   cmMendrelCathodeFrontAxisY.commandConfiguration.offset.offset := 0.0;
   cmMendrelCathodeFrontAxisY.commandConfiguration.offset.profileReference := 1;
   cmMendrelCathodeFrontAxisY.commandConfiguration.offset.offsetDistance := 0.0;
   cmMendrelCathodeFrontAxisY.commandConfiguration.offset.startPosition := 0.0;
   cmMendrelCathodeFrontAxisY.commandConfiguration.offset.direction := 3;
   cmMendrelCathodeFrontAxisY.commandConfiguration.offset.offsetAbsolute := TRUE;
   cmMendrelCathodeFrontAxisY.commandConfiguration.offset.offsetChangeOnTheFly := FALSE;
   cmMendrelCathodeFrontAxisY.commands.enableAxis := FALSE;
   cmMendrelCathodeFrontAxisY.commands.resetAxis := FALSE;
   cmMendrelCathodeFrontAxisY.commands.openBrake := FALSE;
   cmMendrelCathodeFrontAxisY.commands.jogForward := FALSE;
   cmMendrelCathodeFrontAxisY.commands.jogBackward := FALSE;
   cmMendrelCathodeFrontAxisY.commands.moveVelocity := FALSE;
   cmMendrelCathodeFrontAxisY.commands.stop := FALSE;
   cmMendrelCathodeFrontAxisY.commands.fastStop := FALSE;
   cmMendrelCathodeFrontAxisY.commands.torqueLimiting := FALSE;
   cmMendrelCathodeFrontAxisY.commands.homing := FALSE;
   cmMendrelCathodeFrontAxisY.commands.posRelative := FALSE;
   cmMendrelCathodeFrontAxisY.commands.posAbsolute := FALSE;
   cmMendrelCathodeFrontAxisY.commands.posSuperimposed := FALSE;
   cmMendrelCathodeFrontAxisY.commands.haltSuperimposed := FALSE;
   cmMendrelCathodeFrontAxisY.commands.selectSetPosition := -1;
   cmMendrelCathodeFrontAxisY.commands.reset := FALSE;
   cmMendrelCathodeFrontAxisY.monitoring.valid := FALSE;
   cmMendrelCathodeFrontAxisY.monitoring.busy := TRUE;
   cmMendrelCathodeFrontAxisY.monitoring.error := TRUE;
   cmMendrelCathodeFrontAxisY.monitoring.status := 16#8600;
   cmMendrelCathodeFrontAxisY.monitoring.subfunctionStatus := 16#8001;
   cmMendrelCathodeFrontAxisY.monitoring.axisEnabled := FALSE;
   cmMendrelCathodeFrontAxisY.monitoring.resetActive := FALSE;
   cmMendrelCathodeFrontAxisY.monitoring.inVelocity := FALSE;
   cmMendrelCathodeFrontAxisY.monitoring.inLimitation := FALSE;
   cmMendrelCathodeFrontAxisY.monitoring.inClamping := FALSE;
   cmMendrelCathodeFrontAxisY.monitoring.startSync := FALSE;
   cmMendrelCathodeFrontAxisY.monitoring.inSync := FALSE;
   cmMendrelCathodeFrontAxisY.monitoring.inSimulation := FALSE;
   cmMendrelCathodeFrontAxisY.monitoring.jogSelected := FALSE;
   cmMendrelCathodeFrontAxisY.monitoring.moveVelocitySelected := FALSE;
   cmMendrelCathodeFrontAxisY.monitoring.stopSelected := FALSE;
   cmMendrelCathodeFrontAxisY.monitoring.fastStopSelected := FALSE;
   cmMendrelCathodeFrontAxisY.monitoring.torqueLimitingSelected := FALSE;
   cmMendrelCathodeFrontAxisY.monitoring.homingSelected := FALSE;
   cmMendrelCathodeFrontAxisY.monitoring.posRelativeSelected := FALSE;
   cmMendrelCathodeFrontAxisY.monitoring.posAbsoluteSelected := FALSE;
   cmMendrelCathodeFrontAxisY.monitoring.posSuperimposedSelected := FALSE;
   cmMendrelCathodeFrontAxisY.monitoring.haltSuperimposedSelected := FALSE;
   cmMendrelCathodeFrontAxisY.monitoring.commandBusy := FALSE;
   cmMendrelCathodeFrontAxisY.monitoring.commandDone := FALSE;
   cmMendrelCathodeFrontAxisY.monitoring.commandAborted := FALSE;
   cmMendrelCathodeFrontAxisY.monitoring.homingCommandBusy := FALSE;
   cmMendrelCathodeFrontAxisY.monitoring.homingCommandDone := FALSE;
   cmMendrelCathodeFrontAxisY.monitoring.homingCommandAborted := FALSE;
   cmMendrelCathodeFrontAxisY.monitoring.superimposedBusy := FALSE;
   cmMendrelCathodeFrontAxisY.monitoring.superimposedDone := FALSE;
   cmMendrelCathodeFrontAxisY.monitoring.superimposedAborted := FALSE;
   cmMendrelCathodeFrontAxisY.monitoring.actualPosition := 10.963;
   cmMendrelCathodeFrontAxisY.monitoring.actualSpeed := 0.0;
   cmMendrelCathodeFrontAxisY.monitoring.speedUnit := 1062;
   cmMendrelCathodeFrontAxisY.monitoring.positionUnit := 1013;
   cmMendrelCathodeFrontAxisY.monitoring.axisType := 1;
   cmMendrelCathodeFrontAxisY.monitoring.interlockGeneralOut := TRUE;
   cmMendrelCathodeFrontAxisY.monitoring.interlockJogForwardOut := TRUE;
   cmMendrelCathodeFrontAxisY.monitoring.interlockJogBackwardOut := TRUE;
   cmMendrelCathodeFrontAxisZ.commandConfiguration.generalSettings.stopOnError := TRUE;
   cmMendrelCathodeFrontAxisZ.commandConfiguration.generalSettings.resetWithRestart := FALSE;
   cmMendrelCathodeFrontAxisZ.commandConfiguration.generalSettings.abortWaitingSyncCmd := TRUE;
   cmMendrelCathodeFrontAxisZ.commandConfiguration.power.startMode := 1;
   cmMendrelCathodeFrontAxisZ.commandConfiguration.power.stopMode := 0;
   cmMendrelCathodeFrontAxisZ.commandConfiguration.power.syncMotionSimulation := FALSE;
   cmMendrelCathodeFrontAxisZ.commandConfiguration.power.syncMotionSimulationExtendedMode := -1;
   cmMendrelCathodeFrontAxisZ.commandConfiguration.jog.velocity := 5.0;
   cmMendrelCathodeFrontAxisZ.commandConfiguration.jog.acceleration := 50.0;
   cmMendrelCathodeFrontAxisZ.commandConfiguration.jog.deceleration := 50.0;
   cmMendrelCathodeFrontAxisZ.commandConfiguration.jog.jerk := -1.0;
   cmMendrelCathodeFrontAxisZ.commandConfiguration.jog.positionControlled := TRUE;
   cmMendrelCathodeFrontAxisZ.commandConfiguration.jog.increment := 0.0;
   cmMendrelCathodeFrontAxisZ.commandConfiguration.jog.mode := 0;
   cmMendrelCathodeFrontAxisZ.commandConfiguration.moveVelocity.velocity := 0.0;
   cmMendrelCathodeFrontAxisZ.commandConfiguration.moveVelocity.acceleration := -1.0;
   cmMendrelCathodeFrontAxisZ.commandConfiguration.moveVelocity.deceleration := -1.0;
   cmMendrelCathodeFrontAxisZ.commandConfiguration.moveVelocity.jerk := -1.0;
   cmMendrelCathodeFrontAxisZ.commandConfiguration.moveVelocity.direction := 0;
   cmMendrelCathodeFrontAxisZ.commandConfiguration.moveVelocity.positionControlled := TRUE;
   cmMendrelCathodeFrontAxisZ.commandConfiguration.moveVelocity.velocityChangeOnTheFly := FALSE;
   cmMendrelCathodeFrontAxisZ.commandConfiguration.stop.deceleration := -1.0;
   cmMendrelCathodeFrontAxisZ.commandConfiguration.stop.jerk := -1.0;
   cmMendrelCathodeFrontAxisZ.commandConfiguration.stop.abortAcceleration := FALSE;
   cmMendrelCathodeFrontAxisZ.commandConfiguration.fastStop.deceleration := -1.0;
   cmMendrelCathodeFrontAxisZ.commandConfiguration.fastStop.jerk := -1.0;
   cmMendrelCathodeFrontAxisZ.commandConfiguration.fastStop.abortAcceleration := FALSE;
   cmMendrelCathodeFrontAxisZ.commandConfiguration.fastStop.replaceStopPossible := FALSE;
   cmMendrelCathodeFrontAxisZ.commandConfiguration.torqueLimiting.limit := -1.0;
   cmMendrelCathodeFrontAxisZ.commandConfiguration.torqueLimiting.mode := 0;
   cmMendrelCathodeFrontAxisZ.commandConfiguration.homing.position := 0.0;
   cmMendrelCathodeFrontAxisZ.commandConfiguration.homing.mode := 0;
   cmMendrelCathodeFrontAxisZ.commandConfiguration.homing.sensor := 0;
   cmMendrelCathodeFrontAxisZ.commandConfiguration.homing.extendedMode := -1;
   cmMendrelCathodeFrontAxisZ.commandConfiguration.homing.extendedModeTorqueLimit := 0.0;
   cmMendrelCathodeFrontAxisZ.commandConfiguration.homing.extendedModeTargetPosition := 0.0;
   cmMendrelCathodeFrontAxisZ.commandConfiguration.posRelative.distance := 0.0;
   cmMendrelCathodeFrontAxisZ.commandConfiguration.posRelative.velocity := -1.0;
   cmMendrelCathodeFrontAxisZ.commandConfiguration.posRelative.acceleration := -1.0;
   cmMendrelCathodeFrontAxisZ.commandConfiguration.posRelative.deceleration := -1.0;
   cmMendrelCathodeFrontAxisZ.commandConfiguration.posRelative.jerk := -1.0;
   cmMendrelCathodeFrontAxisZ.commandConfiguration.posRelative.direction := 0;
   cmMendrelCathodeFrontAxisZ.commandConfiguration.posAbsolute.position := 0.0;
   cmMendrelCathodeFrontAxisZ.commandConfiguration.posAbsolute.velocity := -1.0;
   cmMendrelCathodeFrontAxisZ.commandConfiguration.posAbsolute.acceleration := -1.0;
   cmMendrelCathodeFrontAxisZ.commandConfiguration.posAbsolute.deceleration := -1.0;
   cmMendrelCathodeFrontAxisZ.commandConfiguration.posAbsolute.jerk := -1.0;
   cmMendrelCathodeFrontAxisZ.commandConfiguration.posAbsolute.direction := 1;
   cmMendrelCathodeFrontAxisZ.commandConfiguration.posAbsolute.positionChangeOnTheFly := FALSE;
   cmMendrelCathodeFrontAxisZ.commandConfiguration.posAbsolute.velocityChangeOnTheFly := FALSE;
   cmMendrelCathodeFrontAxisZ.commandConfiguration.posSuperimposed.distance := 0.0;
   cmMendrelCathodeFrontAxisZ.commandConfiguration.posSuperimposed.velocityDiff := -1.0;
   cmMendrelCathodeFrontAxisZ.commandConfiguration.posSuperimposed.acceleration := -1.0;
   cmMendrelCathodeFrontAxisZ.commandConfiguration.posSuperimposed.deceleration := -1.0;
   cmMendrelCathodeFrontAxisZ.commandConfiguration.posSuperimposed.jerk := -1.0;
   cmMendrelCathodeFrontAxisZ.commandConfiguration.posSuperimposed.direction := 0;
   cmMendrelCathodeFrontAxisZ.commandConfiguration.haltSuperimposed.deceleration := -1.0;
   cmMendrelCathodeFrontAxisZ.commandConfiguration.haltSuperimposed.jerk := -1.0;
   cmMendrelCathodeFrontAxisZ.commandConfiguration.haltSuperimposed.abortAcceleration := FALSE;
   cmMendrelCathodeFrontAxisZ.commandConfiguration.gearInRelative.ratioNumerator := 1;
   cmMendrelCathodeFrontAxisZ.commandConfiguration.gearInRelative.ratioDenominator := 1;
   cmMendrelCathodeFrontAxisZ.commandConfiguration.gearInRelative.acceleration := -1.0;
   cmMendrelCathodeFrontAxisZ.commandConfiguration.gearInRelative.deceleration := -1.0;
   cmMendrelCathodeFrontAxisZ.commandConfiguration.gearInRelative.jerk := -1.0;
   cmMendrelCathodeFrontAxisZ.commandConfiguration.gearInRelative.ratioChangeOnTheFly := FALSE;
   cmMendrelCathodeFrontAxisZ.commandConfiguration.gearInAbsolute.ratioNumerator := 1;
   cmMendrelCathodeFrontAxisZ.commandConfiguration.gearInAbsolute.ratioDenominator := 1;
   cmMendrelCathodeFrontAxisZ.commandConfiguration.gearInAbsolute.masterSyncPosition := 0.0;
   cmMendrelCathodeFrontAxisZ.commandConfiguration.gearInAbsolute.slaveSyncPosition := 0.0;
   cmMendrelCathodeFrontAxisZ.commandConfiguration.gearInAbsolute.syncProfileReference := 1;
   cmMendrelCathodeFrontAxisZ.commandConfiguration.gearInAbsolute.masterStartDistance := 0.0;
   cmMendrelCathodeFrontAxisZ.commandConfiguration.gearInAbsolute.velocity := -1.0;
   cmMendrelCathodeFrontAxisZ.commandConfiguration.gearInAbsolute.acceleration := -1.0;
   cmMendrelCathodeFrontAxisZ.commandConfiguration.gearInAbsolute.deceleration := -1.0;
   cmMendrelCathodeFrontAxisZ.commandConfiguration.gearInAbsolute.jerk := -1.0;
   cmMendrelCathodeFrontAxisZ.commandConfiguration.gearInAbsolute.syncDirection := 1;
   cmMendrelCathodeFrontAxisZ.commandConfiguration.gearInAbsolute.ratioChangeOnTheFly := FALSE;
   cmMendrelCathodeFrontAxisZ.commandConfiguration.gearInVelocity.continuousUpdate := FALSE;
   cmMendrelCathodeFrontAxisZ.commandConfiguration.gearInVelocity.ratioNumerator := 1;
   cmMendrelCathodeFrontAxisZ.commandConfiguration.gearInVelocity.ratioDenominator := 1;
   cmMendrelCathodeFrontAxisZ.commandConfiguration.gearInVelocity.acceleration := -1.0;
   cmMendrelCathodeFrontAxisZ.commandConfiguration.gearInVelocity.deceleration := -1.0;
   cmMendrelCathodeFrontAxisZ.commandConfiguration.gearInVelocity.jerk := -1.0;
   cmMendrelCathodeFrontAxisZ.commandConfiguration.gearInVelocity.positionControlled := FALSE;
   cmMendrelCathodeFrontAxisZ.commandConfiguration.camIn.masterOffset := 0.0;
   cmMendrelCathodeFrontAxisZ.commandConfiguration.camIn.slaveOffset := 0.0;
   cmMendrelCathodeFrontAxisZ.commandConfiguration.camIn.masterScaling := 1.0;
   cmMendrelCathodeFrontAxisZ.commandConfiguration.camIn.slaveScaling := 1.0;
   cmMendrelCathodeFrontAxisZ.commandConfiguration.camIn.masterSyncPosition := 0.0;
   cmMendrelCathodeFrontAxisZ.commandConfiguration.camIn.syncProfileReference := 1;
   cmMendrelCathodeFrontAxisZ.commandConfiguration.camIn.masterStartDistance := 0.0;
   cmMendrelCathodeFrontAxisZ.commandConfiguration.camIn.velocity := -1.0;
   cmMendrelCathodeFrontAxisZ.commandConfiguration.camIn.acceleration := -1.0;
   cmMendrelCathodeFrontAxisZ.commandConfiguration.camIn.deceleration := -1.0;
   cmMendrelCathodeFrontAxisZ.commandConfiguration.camIn.jerk := -1.0;
   cmMendrelCathodeFrontAxisZ.commandConfiguration.camIn.applicationMode := 0;
   cmMendrelCathodeFrontAxisZ.commandConfiguration.camIn.syncDirection := 1;
   cmMendrelCathodeFrontAxisZ.commandConfiguration.gearOutCamOut.slavePosition := 0.0;
   cmMendrelCathodeFrontAxisZ.commandConfiguration.gearOutCamOut.syncProfileReference := 1;
   cmMendrelCathodeFrontAxisZ.commandConfiguration.gearOutCamOut.masterStopDistance := 0.0;
   cmMendrelCathodeFrontAxisZ.commandConfiguration.gearOutCamOut.deceleration := -1.0;
   cmMendrelCathodeFrontAxisZ.commandConfiguration.gearOutCamOut.jerk := -1.0;
   cmMendrelCathodeFrontAxisZ.commandConfiguration.gearOutCamOut.syncOutDirection := 3;
   cmMendrelCathodeFrontAxisZ.commandConfiguration.gearOutCamOut.gearOutCamOutMode := -1;
   cmMendrelCathodeFrontAxisZ.commandConfiguration.phasing.phaseShift := 0.0;
   cmMendrelCathodeFrontAxisZ.commandConfiguration.phasing.velocity := -1.0;
   cmMendrelCathodeFrontAxisZ.commandConfiguration.phasing.acceleration := -1.0;
   cmMendrelCathodeFrontAxisZ.commandConfiguration.phasing.deceleration := -1.0;
   cmMendrelCathodeFrontAxisZ.commandConfiguration.phasing.jerk := -1.0;
   cmMendrelCathodeFrontAxisZ.commandConfiguration.phasing.profileReference := 0;
   cmMendrelCathodeFrontAxisZ.commandConfiguration.phasing.phasingDistance := 0.0;
   cmMendrelCathodeFrontAxisZ.commandConfiguration.phasing.startPosition := 0.0;
   cmMendrelCathodeFrontAxisZ.commandConfiguration.phasing.direction := 3;
   cmMendrelCathodeFrontAxisZ.commandConfiguration.phasing.phaseAbsolute := TRUE;
   cmMendrelCathodeFrontAxisZ.commandConfiguration.phasing.phaseShiftChangeOnTheFly := FALSE;
   cmMendrelCathodeFrontAxisZ.commandConfiguration.offset.offset := 0.0;
   cmMendrelCathodeFrontAxisZ.commandConfiguration.offset.profileReference := 1;
   cmMendrelCathodeFrontAxisZ.commandConfiguration.offset.offsetDistance := 0.0;
   cmMendrelCathodeFrontAxisZ.commandConfiguration.offset.startPosition := 0.0;
   cmMendrelCathodeFrontAxisZ.commandConfiguration.offset.direction := 3;
   cmMendrelCathodeFrontAxisZ.commandConfiguration.offset.offsetAbsolute := TRUE;
   cmMendrelCathodeFrontAxisZ.commandConfiguration.offset.offsetChangeOnTheFly := FALSE;
   cmMendrelCathodeFrontAxisZ.commands.enableAxis := FALSE;
   cmMendrelCathodeFrontAxisZ.commands.resetAxis := FALSE;
   cmMendrelCathodeFrontAxisZ.commands.openBrake := FALSE;
   cmMendrelCathodeFrontAxisZ.commands.jogForward := FALSE;
   cmMendrelCathodeFrontAxisZ.commands.jogBackward := FALSE;
   cmMendrelCathodeFrontAxisZ.commands.moveVelocity := FALSE;
   cmMendrelCathodeFrontAxisZ.commands.stop := FALSE;
   cmMendrelCathodeFrontAxisZ.commands.fastStop := FALSE;
   cmMendrelCathodeFrontAxisZ.commands.torqueLimiting := FALSE;
   cmMendrelCathodeFrontAxisZ.commands.homing := FALSE;
   cmMendrelCathodeFrontAxisZ.commands.posRelative := FALSE;
   cmMendrelCathodeFrontAxisZ.commands.posAbsolute := FALSE;
   cmMendrelCathodeFrontAxisZ.commands.posSuperimposed := FALSE;
   cmMendrelCathodeFrontAxisZ.commands.haltSuperimposed := FALSE;
   cmMendrelCathodeFrontAxisZ.commands.selectSetPosition := -1;
   cmMendrelCathodeFrontAxisZ.commands.reset := FALSE;
   cmMendrelCathodeFrontAxisZ.monitoring.valid := FALSE;
   cmMendrelCathodeFrontAxisZ.monitoring.busy := TRUE;
   cmMendrelCathodeFrontAxisZ.monitoring.error := TRUE;
   cmMendrelCathodeFrontAxisZ.monitoring.status := 16#8600;
   cmMendrelCathodeFrontAxisZ.monitoring.subfunctionStatus := 16#8001;
   cmMendrelCathodeFrontAxisZ.monitoring.axisEnabled := FALSE;
   cmMendrelCathodeFrontAxisZ.monitoring.resetActive := FALSE;
   cmMendrelCathodeFrontAxisZ.monitoring.inVelocity := FALSE;
   cmMendrelCathodeFrontAxisZ.monitoring.inLimitation := FALSE;
   cmMendrelCathodeFrontAxisZ.monitoring.inClamping := FALSE;
   cmMendrelCathodeFrontAxisZ.monitoring.startSync := FALSE;
   cmMendrelCathodeFrontAxisZ.monitoring.inSync := FALSE;
   cmMendrelCathodeFrontAxisZ.monitoring.inSimulation := FALSE;
   cmMendrelCathodeFrontAxisZ.monitoring.jogSelected := FALSE;
   cmMendrelCathodeFrontAxisZ.monitoring.moveVelocitySelected := FALSE;
   cmMendrelCathodeFrontAxisZ.monitoring.stopSelected := FALSE;
   cmMendrelCathodeFrontAxisZ.monitoring.fastStopSelected := FALSE;
   cmMendrelCathodeFrontAxisZ.monitoring.torqueLimitingSelected := FALSE;
   cmMendrelCathodeFrontAxisZ.monitoring.homingSelected := FALSE;
   cmMendrelCathodeFrontAxisZ.monitoring.posRelativeSelected := FALSE;
   cmMendrelCathodeFrontAxisZ.monitoring.posAbsoluteSelected := FALSE;
   cmMendrelCathodeFrontAxisZ.monitoring.posSuperimposedSelected := FALSE;
   cmMendrelCathodeFrontAxisZ.monitoring.haltSuperimposedSelected := FALSE;
   cmMendrelCathodeFrontAxisZ.monitoring.commandBusy := FALSE;
   cmMendrelCathodeFrontAxisZ.monitoring.commandDone := FALSE;
   cmMendrelCathodeFrontAxisZ.monitoring.commandAborted := FALSE;
   cmMendrelCathodeFrontAxisZ.monitoring.homingCommandBusy := FALSE;
   cmMendrelCathodeFrontAxisZ.monitoring.homingCommandDone := FALSE;
   cmMendrelCathodeFrontAxisZ.monitoring.homingCommandAborted := FALSE;
   cmMendrelCathodeFrontAxisZ.monitoring.superimposedBusy := FALSE;
   cmMendrelCathodeFrontAxisZ.monitoring.superimposedDone := FALSE;
   cmMendrelCathodeFrontAxisZ.monitoring.superimposedAborted := FALSE;
   cmMendrelCathodeFrontAxisZ.monitoring.actualPosition := 13.099;
   cmMendrelCathodeFrontAxisZ.monitoring.actualSpeed := 0.0;
   cmMendrelCathodeFrontAxisZ.monitoring.speedUnit := 1062;
   cmMendrelCathodeFrontAxisZ.monitoring.positionUnit := 1013;
   cmMendrelCathodeFrontAxisZ.monitoring.axisType := 1;
   cmMendrelCathodeFrontAxisZ.monitoring.interlockGeneralOut := TRUE;
   cmMendrelCathodeFrontAxisZ.monitoring.interlockJogForwardOut := TRUE;
   cmMendrelCathodeFrontAxisZ.monitoring.interlockJogBackwardOut := TRUE;
   cmMendrelCathodeRearAxisY.commandConfiguration.generalSettings.stopOnError := TRUE;
   cmMendrelCathodeRearAxisY.commandConfiguration.generalSettings.resetWithRestart := FALSE;
   cmMendrelCathodeRearAxisY.commandConfiguration.generalSettings.abortWaitingSyncCmd := TRUE;
   cmMendrelCathodeRearAxisY.commandConfiguration.power.startMode := 1;
   cmMendrelCathodeRearAxisY.commandConfiguration.power.stopMode := 0;
   cmMendrelCathodeRearAxisY.commandConfiguration.power.syncMotionSimulation := FALSE;
   cmMendrelCathodeRearAxisY.commandConfiguration.power.syncMotionSimulationExtendedMode := -1;
   cmMendrelCathodeRearAxisY.commandConfiguration.jog.velocity := 0.0;
   cmMendrelCathodeRearAxisY.commandConfiguration.jog.acceleration := -1.0;
   cmMendrelCathodeRearAxisY.commandConfiguration.jog.deceleration := -1.0;
   cmMendrelCathodeRearAxisY.commandConfiguration.jog.jerk := -1.0;
   cmMendrelCathodeRearAxisY.commandConfiguration.jog.positionControlled := TRUE;
   cmMendrelCathodeRearAxisY.commandConfiguration.jog.increment := 0.0;
   cmMendrelCathodeRearAxisY.commandConfiguration.jog.mode := 0;
   cmMendrelCathodeRearAxisY.commandConfiguration.moveVelocity.velocity := 0.0;
   cmMendrelCathodeRearAxisY.commandConfiguration.moveVelocity.acceleration := -1.0;
   cmMendrelCathodeRearAxisY.commandConfiguration.moveVelocity.deceleration := -1.0;
   cmMendrelCathodeRearAxisY.commandConfiguration.moveVelocity.jerk := -1.0;
   cmMendrelCathodeRearAxisY.commandConfiguration.moveVelocity.direction := 0;
   cmMendrelCathodeRearAxisY.commandConfiguration.moveVelocity.positionControlled := TRUE;
   cmMendrelCathodeRearAxisY.commandConfiguration.moveVelocity.velocityChangeOnTheFly := FALSE;
   cmMendrelCathodeRearAxisY.commandConfiguration.stop.deceleration := -1.0;
   cmMendrelCathodeRearAxisY.commandConfiguration.stop.jerk := -1.0;
   cmMendrelCathodeRearAxisY.commandConfiguration.stop.abortAcceleration := FALSE;
   cmMendrelCathodeRearAxisY.commandConfiguration.fastStop.deceleration := -1.0;
   cmMendrelCathodeRearAxisY.commandConfiguration.fastStop.jerk := -1.0;
   cmMendrelCathodeRearAxisY.commandConfiguration.fastStop.abortAcceleration := FALSE;
   cmMendrelCathodeRearAxisY.commandConfiguration.fastStop.replaceStopPossible := FALSE;
   cmMendrelCathodeRearAxisY.commandConfiguration.torqueLimiting.limit := -1.0;
   cmMendrelCathodeRearAxisY.commandConfiguration.torqueLimiting.mode := 0;
   cmMendrelCathodeRearAxisY.commandConfiguration.homing.position := 0.0;
   cmMendrelCathodeRearAxisY.commandConfiguration.homing.mode := 0;
   cmMendrelCathodeRearAxisY.commandConfiguration.homing.sensor := 0;
   cmMendrelCathodeRearAxisY.commandConfiguration.homing.extendedMode := -1;
   cmMendrelCathodeRearAxisY.commandConfiguration.homing.extendedModeTorqueLimit := 0.0;
   cmMendrelCathodeRearAxisY.commandConfiguration.homing.extendedModeTargetPosition := 0.0;
   cmMendrelCathodeRearAxisY.commandConfiguration.posRelative.distance := 0.0;
   cmMendrelCathodeRearAxisY.commandConfiguration.posRelative.velocity := -1.0;
   cmMendrelCathodeRearAxisY.commandConfiguration.posRelative.acceleration := -1.0;
   cmMendrelCathodeRearAxisY.commandConfiguration.posRelative.deceleration := -1.0;
   cmMendrelCathodeRearAxisY.commandConfiguration.posRelative.jerk := -1.0;
   cmMendrelCathodeRearAxisY.commandConfiguration.posRelative.direction := 0;
   cmMendrelCathodeRearAxisY.commandConfiguration.posAbsolute.position := 0.0;
   cmMendrelCathodeRearAxisY.commandConfiguration.posAbsolute.velocity := -1.0;
   cmMendrelCathodeRearAxisY.commandConfiguration.posAbsolute.acceleration := -1.0;
   cmMendrelCathodeRearAxisY.commandConfiguration.posAbsolute.deceleration := -1.0;
   cmMendrelCathodeRearAxisY.commandConfiguration.posAbsolute.jerk := -1.0;
   cmMendrelCathodeRearAxisY.commandConfiguration.posAbsolute.direction := 1;
   cmMendrelCathodeRearAxisY.commandConfiguration.posAbsolute.positionChangeOnTheFly := FALSE;
   cmMendrelCathodeRearAxisY.commandConfiguration.posAbsolute.velocityChangeOnTheFly := FALSE;
   cmMendrelCathodeRearAxisY.commandConfiguration.posSuperimposed.distance := 0.0;
   cmMendrelCathodeRearAxisY.commandConfiguration.posSuperimposed.velocityDiff := -1.0;
   cmMendrelCathodeRearAxisY.commandConfiguration.posSuperimposed.acceleration := -1.0;
   cmMendrelCathodeRearAxisY.commandConfiguration.posSuperimposed.deceleration := -1.0;
   cmMendrelCathodeRearAxisY.commandConfiguration.posSuperimposed.jerk := -1.0;
   cmMendrelCathodeRearAxisY.commandConfiguration.posSuperimposed.direction := 0;
   cmMendrelCathodeRearAxisY.commandConfiguration.haltSuperimposed.deceleration := -1.0;
   cmMendrelCathodeRearAxisY.commandConfiguration.haltSuperimposed.jerk := -1.0;
   cmMendrelCathodeRearAxisY.commandConfiguration.haltSuperimposed.abortAcceleration := FALSE;
   cmMendrelCathodeRearAxisY.commandConfiguration.gearInRelative.ratioNumerator := 1;
   cmMendrelCathodeRearAxisY.commandConfiguration.gearInRelative.ratioDenominator := 1;
   cmMendrelCathodeRearAxisY.commandConfiguration.gearInRelative.acceleration := -1.0;
   cmMendrelCathodeRearAxisY.commandConfiguration.gearInRelative.deceleration := -1.0;
   cmMendrelCathodeRearAxisY.commandConfiguration.gearInRelative.jerk := -1.0;
   cmMendrelCathodeRearAxisY.commandConfiguration.gearInRelative.ratioChangeOnTheFly := FALSE;
   cmMendrelCathodeRearAxisY.commandConfiguration.gearInAbsolute.ratioNumerator := 1;
   cmMendrelCathodeRearAxisY.commandConfiguration.gearInAbsolute.ratioDenominator := 1;
   cmMendrelCathodeRearAxisY.commandConfiguration.gearInAbsolute.masterSyncPosition := 0.0;
   cmMendrelCathodeRearAxisY.commandConfiguration.gearInAbsolute.slaveSyncPosition := 0.0;
   cmMendrelCathodeRearAxisY.commandConfiguration.gearInAbsolute.syncProfileReference := 1;
   cmMendrelCathodeRearAxisY.commandConfiguration.gearInAbsolute.masterStartDistance := 0.0;
   cmMendrelCathodeRearAxisY.commandConfiguration.gearInAbsolute.velocity := -1.0;
   cmMendrelCathodeRearAxisY.commandConfiguration.gearInAbsolute.acceleration := -1.0;
   cmMendrelCathodeRearAxisY.commandConfiguration.gearInAbsolute.deceleration := -1.0;
   cmMendrelCathodeRearAxisY.commandConfiguration.gearInAbsolute.jerk := -1.0;
   cmMendrelCathodeRearAxisY.commandConfiguration.gearInAbsolute.syncDirection := 1;
   cmMendrelCathodeRearAxisY.commandConfiguration.gearInAbsolute.ratioChangeOnTheFly := FALSE;
   cmMendrelCathodeRearAxisY.commandConfiguration.gearInVelocity.continuousUpdate := FALSE;
   cmMendrelCathodeRearAxisY.commandConfiguration.gearInVelocity.ratioNumerator := 1;
   cmMendrelCathodeRearAxisY.commandConfiguration.gearInVelocity.ratioDenominator := 1;
   cmMendrelCathodeRearAxisY.commandConfiguration.gearInVelocity.acceleration := -1.0;
   cmMendrelCathodeRearAxisY.commandConfiguration.gearInVelocity.deceleration := -1.0;
   cmMendrelCathodeRearAxisY.commandConfiguration.gearInVelocity.jerk := -1.0;
   cmMendrelCathodeRearAxisY.commandConfiguration.gearInVelocity.positionControlled := FALSE;
   cmMendrelCathodeRearAxisY.commandConfiguration.camIn.masterOffset := 0.0;
   cmMendrelCathodeRearAxisY.commandConfiguration.camIn.slaveOffset := 0.0;
   cmMendrelCathodeRearAxisY.commandConfiguration.camIn.masterScaling := 1.0;
   cmMendrelCathodeRearAxisY.commandConfiguration.camIn.slaveScaling := 1.0;
   cmMendrelCathodeRearAxisY.commandConfiguration.camIn.masterSyncPosition := 0.0;
   cmMendrelCathodeRearAxisY.commandConfiguration.camIn.syncProfileReference := 1;
   cmMendrelCathodeRearAxisY.commandConfiguration.camIn.masterStartDistance := 0.0;
   cmMendrelCathodeRearAxisY.commandConfiguration.camIn.velocity := -1.0;
   cmMendrelCathodeRearAxisY.commandConfiguration.camIn.acceleration := -1.0;
   cmMendrelCathodeRearAxisY.commandConfiguration.camIn.deceleration := -1.0;
   cmMendrelCathodeRearAxisY.commandConfiguration.camIn.jerk := -1.0;
   cmMendrelCathodeRearAxisY.commandConfiguration.camIn.applicationMode := 0;
   cmMendrelCathodeRearAxisY.commandConfiguration.camIn.syncDirection := 1;
   cmMendrelCathodeRearAxisY.commandConfiguration.gearOutCamOut.slavePosition := 0.0;
   cmMendrelCathodeRearAxisY.commandConfiguration.gearOutCamOut.syncProfileReference := 1;
   cmMendrelCathodeRearAxisY.commandConfiguration.gearOutCamOut.masterStopDistance := 0.0;
   cmMendrelCathodeRearAxisY.commandConfiguration.gearOutCamOut.deceleration := -1.0;
   cmMendrelCathodeRearAxisY.commandConfiguration.gearOutCamOut.jerk := -1.0;
   cmMendrelCathodeRearAxisY.commandConfiguration.gearOutCamOut.syncOutDirection := 3;
   cmMendrelCathodeRearAxisY.commandConfiguration.gearOutCamOut.gearOutCamOutMode := -1;
   cmMendrelCathodeRearAxisY.commandConfiguration.phasing.phaseShift := 0.0;
   cmMendrelCathodeRearAxisY.commandConfiguration.phasing.velocity := -1.0;
   cmMendrelCathodeRearAxisY.commandConfiguration.phasing.acceleration := -1.0;
   cmMendrelCathodeRearAxisY.commandConfiguration.phasing.deceleration := -1.0;
   cmMendrelCathodeRearAxisY.commandConfiguration.phasing.jerk := -1.0;
   cmMendrelCathodeRearAxisY.commandConfiguration.phasing.profileReference := 0;
   cmMendrelCathodeRearAxisY.commandConfiguration.phasing.phasingDistance := 0.0;
   cmMendrelCathodeRearAxisY.commandConfiguration.phasing.startPosition := 0.0;
   cmMendrelCathodeRearAxisY.commandConfiguration.phasing.direction := 3;
   cmMendrelCathodeRearAxisY.commandConfiguration.phasing.phaseAbsolute := TRUE;
   cmMendrelCathodeRearAxisY.commandConfiguration.phasing.phaseShiftChangeOnTheFly := FALSE;
   cmMendrelCathodeRearAxisY.commandConfiguration.offset.offset := 0.0;
   cmMendrelCathodeRearAxisY.commandConfiguration.offset.profileReference := 1;
   cmMendrelCathodeRearAxisY.commandConfiguration.offset.offsetDistance := 0.0;
   cmMendrelCathodeRearAxisY.commandConfiguration.offset.startPosition := 0.0;
   cmMendrelCathodeRearAxisY.commandConfiguration.offset.direction := 3;
   cmMendrelCathodeRearAxisY.commandConfiguration.offset.offsetAbsolute := TRUE;
   cmMendrelCathodeRearAxisY.commandConfiguration.offset.offsetChangeOnTheFly := FALSE;
   cmMendrelCathodeRearAxisY.commands.enableAxis := FALSE;
   cmMendrelCathodeRearAxisY.commands.resetAxis := FALSE;
   cmMendrelCathodeRearAxisY.commands.openBrake := FALSE;
   cmMendrelCathodeRearAxisY.commands.jogForward := FALSE;
   cmMendrelCathodeRearAxisY.commands.jogBackward := FALSE;
   cmMendrelCathodeRearAxisY.commands.moveVelocity := FALSE;
   cmMendrelCathodeRearAxisY.commands.stop := FALSE;
   cmMendrelCathodeRearAxisY.commands.fastStop := FALSE;
   cmMendrelCathodeRearAxisY.commands.torqueLimiting := FALSE;
   cmMendrelCathodeRearAxisY.commands.homing := FALSE;
   cmMendrelCathodeRearAxisY.commands.posRelative := FALSE;
   cmMendrelCathodeRearAxisY.commands.posAbsolute := FALSE;
   cmMendrelCathodeRearAxisY.commands.posSuperimposed := FALSE;
   cmMendrelCathodeRearAxisY.commands.haltSuperimposed := FALSE;
   cmMendrelCathodeRearAxisY.commands.selectSetPosition := -1;
   cmMendrelCathodeRearAxisY.commands.reset := FALSE;
   cmMendrelCathodeRearAxisY.monitoring.valid := FALSE;
   cmMendrelCathodeRearAxisY.monitoring.busy := TRUE;
   cmMendrelCathodeRearAxisY.monitoring.error := TRUE;
   cmMendrelCathodeRearAxisY.monitoring.status := 16#8600;
   cmMendrelCathodeRearAxisY.monitoring.subfunctionStatus := 16#8001;
   cmMendrelCathodeRearAxisY.monitoring.axisEnabled := FALSE;
   cmMendrelCathodeRearAxisY.monitoring.resetActive := FALSE;
   cmMendrelCathodeRearAxisY.monitoring.inVelocity := FALSE;
   cmMendrelCathodeRearAxisY.monitoring.inLimitation := FALSE;
   cmMendrelCathodeRearAxisY.monitoring.inClamping := FALSE;
   cmMendrelCathodeRearAxisY.monitoring.startSync := FALSE;
   cmMendrelCathodeRearAxisY.monitoring.inSync := FALSE;
   cmMendrelCathodeRearAxisY.monitoring.inSimulation := FALSE;
   cmMendrelCathodeRearAxisY.monitoring.jogSelected := FALSE;
   cmMendrelCathodeRearAxisY.monitoring.moveVelocitySelected := FALSE;
   cmMendrelCathodeRearAxisY.monitoring.stopSelected := FALSE;
   cmMendrelCathodeRearAxisY.monitoring.fastStopSelected := FALSE;
   cmMendrelCathodeRearAxisY.monitoring.torqueLimitingSelected := FALSE;
   cmMendrelCathodeRearAxisY.monitoring.homingSelected := FALSE;
   cmMendrelCathodeRearAxisY.monitoring.posRelativeSelected := FALSE;
   cmMendrelCathodeRearAxisY.monitoring.posAbsoluteSelected := FALSE;
   cmMendrelCathodeRearAxisY.monitoring.posSuperimposedSelected := FALSE;
   cmMendrelCathodeRearAxisY.monitoring.haltSuperimposedSelected := FALSE;
   cmMendrelCathodeRearAxisY.monitoring.commandBusy := FALSE;
   cmMendrelCathodeRearAxisY.monitoring.commandDone := FALSE;
   cmMendrelCathodeRearAxisY.monitoring.commandAborted := FALSE;
   cmMendrelCathodeRearAxisY.monitoring.homingCommandBusy := FALSE;
   cmMendrelCathodeRearAxisY.monitoring.homingCommandDone := FALSE;
   cmMendrelCathodeRearAxisY.monitoring.homingCommandAborted := FALSE;
   cmMendrelCathodeRearAxisY.monitoring.superimposedBusy := FALSE;
   cmMendrelCathodeRearAxisY.monitoring.superimposedDone := FALSE;
   cmMendrelCathodeRearAxisY.monitoring.superimposedAborted := FALSE;
   cmMendrelCathodeRearAxisY.monitoring.actualPosition := 12.417;
   cmMendrelCathodeRearAxisY.monitoring.actualSpeed := 0.0;
   cmMendrelCathodeRearAxisY.monitoring.speedUnit := 1062;
   cmMendrelCathodeRearAxisY.monitoring.positionUnit := 1013;
   cmMendrelCathodeRearAxisY.monitoring.axisType := 1;
   cmMendrelCathodeRearAxisY.monitoring.interlockGeneralOut := TRUE;
   cmMendrelCathodeRearAxisY.monitoring.interlockJogForwardOut := TRUE;
   cmMendrelCathodeRearAxisY.monitoring.interlockJogBackwardOut := TRUE;
   cmMendrelCathodeRearAxisZ.commandConfiguration.generalSettings.stopOnError := TRUE;
   cmMendrelCathodeRearAxisZ.commandConfiguration.generalSettings.resetWithRestart := FALSE;
   cmMendrelCathodeRearAxisZ.commandConfiguration.generalSettings.abortWaitingSyncCmd := TRUE;
   cmMendrelCathodeRearAxisZ.commandConfiguration.power.startMode := 1;
   cmMendrelCathodeRearAxisZ.commandConfiguration.power.stopMode := 0;
   cmMendrelCathodeRearAxisZ.commandConfiguration.power.syncMotionSimulation := FALSE;
   cmMendrelCathodeRearAxisZ.commandConfiguration.power.syncMotionSimulationExtendedMode := -1;
   cmMendrelCathodeRearAxisZ.commandConfiguration.jog.velocity := 0.0;
   cmMendrelCathodeRearAxisZ.commandConfiguration.jog.acceleration := -1.0;
   cmMendrelCathodeRearAxisZ.commandConfiguration.jog.deceleration := -1.0;
   cmMendrelCathodeRearAxisZ.commandConfiguration.jog.jerk := -1.0;
   cmMendrelCathodeRearAxisZ.commandConfiguration.jog.positionControlled := TRUE;
   cmMendrelCathodeRearAxisZ.commandConfiguration.jog.increment := 0.0;
   cmMendrelCathodeRearAxisZ.commandConfiguration.jog.mode := 0;
   cmMendrelCathodeRearAxisZ.commandConfiguration.moveVelocity.velocity := 0.0;
   cmMendrelCathodeRearAxisZ.commandConfiguration.moveVelocity.acceleration := -1.0;
   cmMendrelCathodeRearAxisZ.commandConfiguration.moveVelocity.deceleration := -1.0;
   cmMendrelCathodeRearAxisZ.commandConfiguration.moveVelocity.jerk := -1.0;
   cmMendrelCathodeRearAxisZ.commandConfiguration.moveVelocity.direction := 0;
   cmMendrelCathodeRearAxisZ.commandConfiguration.moveVelocity.positionControlled := TRUE;
   cmMendrelCathodeRearAxisZ.commandConfiguration.moveVelocity.velocityChangeOnTheFly := FALSE;
   cmMendrelCathodeRearAxisZ.commandConfiguration.stop.deceleration := -1.0;
   cmMendrelCathodeRearAxisZ.commandConfiguration.stop.jerk := -1.0;
   cmMendrelCathodeRearAxisZ.commandConfiguration.stop.abortAcceleration := FALSE;
   cmMendrelCathodeRearAxisZ.commandConfiguration.fastStop.deceleration := -1.0;
   cmMendrelCathodeRearAxisZ.commandConfiguration.fastStop.jerk := -1.0;
   cmMendrelCathodeRearAxisZ.commandConfiguration.fastStop.abortAcceleration := FALSE;
   cmMendrelCathodeRearAxisZ.commandConfiguration.fastStop.replaceStopPossible := FALSE;
   cmMendrelCathodeRearAxisZ.commandConfiguration.torqueLimiting.limit := -1.0;
   cmMendrelCathodeRearAxisZ.commandConfiguration.torqueLimiting.mode := 0;
   cmMendrelCathodeRearAxisZ.commandConfiguration.homing.position := 0.0;
   cmMendrelCathodeRearAxisZ.commandConfiguration.homing.mode := 0;
   cmMendrelCathodeRearAxisZ.commandConfiguration.homing.sensor := 0;
   cmMendrelCathodeRearAxisZ.commandConfiguration.homing.extendedMode := -1;
   cmMendrelCathodeRearAxisZ.commandConfiguration.homing.extendedModeTorqueLimit := 0.0;
   cmMendrelCathodeRearAxisZ.commandConfiguration.homing.extendedModeTargetPosition := 0.0;
   cmMendrelCathodeRearAxisZ.commandConfiguration.posRelative.distance := 0.0;
   cmMendrelCathodeRearAxisZ.commandConfiguration.posRelative.velocity := -1.0;
   cmMendrelCathodeRearAxisZ.commandConfiguration.posRelative.acceleration := -1.0;
   cmMendrelCathodeRearAxisZ.commandConfiguration.posRelative.deceleration := -1.0;
   cmMendrelCathodeRearAxisZ.commandConfiguration.posRelative.jerk := -1.0;
   cmMendrelCathodeRearAxisZ.commandConfiguration.posRelative.direction := 0;
   cmMendrelCathodeRearAxisZ.commandConfiguration.posAbsolute.position := 0.0;
   cmMendrelCathodeRearAxisZ.commandConfiguration.posAbsolute.velocity := -1.0;
   cmMendrelCathodeRearAxisZ.commandConfiguration.posAbsolute.acceleration := -1.0;
   cmMendrelCathodeRearAxisZ.commandConfiguration.posAbsolute.deceleration := -1.0;
   cmMendrelCathodeRearAxisZ.commandConfiguration.posAbsolute.jerk := -1.0;
   cmMendrelCathodeRearAxisZ.commandConfiguration.posAbsolute.direction := 1;
   cmMendrelCathodeRearAxisZ.commandConfiguration.posAbsolute.positionChangeOnTheFly := FALSE;
   cmMendrelCathodeRearAxisZ.commandConfiguration.posAbsolute.velocityChangeOnTheFly := FALSE;
   cmMendrelCathodeRearAxisZ.commandConfiguration.posSuperimposed.distance := 0.0;
   cmMendrelCathodeRearAxisZ.commandConfiguration.posSuperimposed.velocityDiff := -1.0;
   cmMendrelCathodeRearAxisZ.commandConfiguration.posSuperimposed.acceleration := -1.0;
   cmMendrelCathodeRearAxisZ.commandConfiguration.posSuperimposed.deceleration := -1.0;
   cmMendrelCathodeRearAxisZ.commandConfiguration.posSuperimposed.jerk := -1.0;
   cmMendrelCathodeRearAxisZ.commandConfiguration.posSuperimposed.direction := 0;
   cmMendrelCathodeRearAxisZ.commandConfiguration.haltSuperimposed.deceleration := -1.0;
   cmMendrelCathodeRearAxisZ.commandConfiguration.haltSuperimposed.jerk := -1.0;
   cmMendrelCathodeRearAxisZ.commandConfiguration.haltSuperimposed.abortAcceleration := FALSE;
   cmMendrelCathodeRearAxisZ.commandConfiguration.gearInRelative.ratioNumerator := 1;
   cmMendrelCathodeRearAxisZ.commandConfiguration.gearInRelative.ratioDenominator := 1;
   cmMendrelCathodeRearAxisZ.commandConfiguration.gearInRelative.acceleration := -1.0;
   cmMendrelCathodeRearAxisZ.commandConfiguration.gearInRelative.deceleration := -1.0;
   cmMendrelCathodeRearAxisZ.commandConfiguration.gearInRelative.jerk := -1.0;
   cmMendrelCathodeRearAxisZ.commandConfiguration.gearInRelative.ratioChangeOnTheFly := FALSE;
   cmMendrelCathodeRearAxisZ.commandConfiguration.gearInAbsolute.ratioNumerator := 1;
   cmMendrelCathodeRearAxisZ.commandConfiguration.gearInAbsolute.ratioDenominator := 1;
   cmMendrelCathodeRearAxisZ.commandConfiguration.gearInAbsolute.masterSyncPosition := 0.0;
   cmMendrelCathodeRearAxisZ.commandConfiguration.gearInAbsolute.slaveSyncPosition := 0.0;
   cmMendrelCathodeRearAxisZ.commandConfiguration.gearInAbsolute.syncProfileReference := 1;
   cmMendrelCathodeRearAxisZ.commandConfiguration.gearInAbsolute.masterStartDistance := 0.0;
   cmMendrelCathodeRearAxisZ.commandConfiguration.gearInAbsolute.velocity := -1.0;
   cmMendrelCathodeRearAxisZ.commandConfiguration.gearInAbsolute.acceleration := -1.0;
   cmMendrelCathodeRearAxisZ.commandConfiguration.gearInAbsolute.deceleration := -1.0;
   cmMendrelCathodeRearAxisZ.commandConfiguration.gearInAbsolute.jerk := -1.0;
   cmMendrelCathodeRearAxisZ.commandConfiguration.gearInAbsolute.syncDirection := 1;
   cmMendrelCathodeRearAxisZ.commandConfiguration.gearInAbsolute.ratioChangeOnTheFly := FALSE;
   cmMendrelCathodeRearAxisZ.commandConfiguration.gearInVelocity.continuousUpdate := FALSE;
   cmMendrelCathodeRearAxisZ.commandConfiguration.gearInVelocity.ratioNumerator := 1;
   cmMendrelCathodeRearAxisZ.commandConfiguration.gearInVelocity.ratioDenominator := 1;
   cmMendrelCathodeRearAxisZ.commandConfiguration.gearInVelocity.acceleration := -1.0;
   cmMendrelCathodeRearAxisZ.commandConfiguration.gearInVelocity.deceleration := -1.0;
   cmMendrelCathodeRearAxisZ.commandConfiguration.gearInVelocity.jerk := -1.0;
   cmMendrelCathodeRearAxisZ.commandConfiguration.gearInVelocity.positionControlled := FALSE;
   cmMendrelCathodeRearAxisZ.commandConfiguration.camIn.masterOffset := 0.0;
   cmMendrelCathodeRearAxisZ.commandConfiguration.camIn.slaveOffset := 0.0;
   cmMendrelCathodeRearAxisZ.commandConfiguration.camIn.masterScaling := 1.0;
   cmMendrelCathodeRearAxisZ.commandConfiguration.camIn.slaveScaling := 1.0;
   cmMendrelCathodeRearAxisZ.commandConfiguration.camIn.masterSyncPosition := 0.0;
   cmMendrelCathodeRearAxisZ.commandConfiguration.camIn.syncProfileReference := 1;
   cmMendrelCathodeRearAxisZ.commandConfiguration.camIn.masterStartDistance := 0.0;
   cmMendrelCathodeRearAxisZ.commandConfiguration.camIn.velocity := -1.0;
   cmMendrelCathodeRearAxisZ.commandConfiguration.camIn.acceleration := -1.0;
   cmMendrelCathodeRearAxisZ.commandConfiguration.camIn.deceleration := -1.0;
   cmMendrelCathodeRearAxisZ.commandConfiguration.camIn.jerk := -1.0;
   cmMendrelCathodeRearAxisZ.commandConfiguration.camIn.applicationMode := 0;
   cmMendrelCathodeRearAxisZ.commandConfiguration.camIn.syncDirection := 1;
   cmMendrelCathodeRearAxisZ.commandConfiguration.gearOutCamOut.slavePosition := 0.0;
   cmMendrelCathodeRearAxisZ.commandConfiguration.gearOutCamOut.syncProfileReference := 1;
   cmMendrelCathodeRearAxisZ.commandConfiguration.gearOutCamOut.masterStopDistance := 0.0;
   cmMendrelCathodeRearAxisZ.commandConfiguration.gearOutCamOut.deceleration := -1.0;
   cmMendrelCathodeRearAxisZ.commandConfiguration.gearOutCamOut.jerk := -1.0;
   cmMendrelCathodeRearAxisZ.commandConfiguration.gearOutCamOut.syncOutDirection := 3;
   cmMendrelCathodeRearAxisZ.commandConfiguration.gearOutCamOut.gearOutCamOutMode := -1;
   cmMendrelCathodeRearAxisZ.commandConfiguration.phasing.phaseShift := 0.0;
   cmMendrelCathodeRearAxisZ.commandConfiguration.phasing.velocity := -1.0;
   cmMendrelCathodeRearAxisZ.commandConfiguration.phasing.acceleration := -1.0;
   cmMendrelCathodeRearAxisZ.commandConfiguration.phasing.deceleration := -1.0;
   cmMendrelCathodeRearAxisZ.commandConfiguration.phasing.jerk := -1.0;
   cmMendrelCathodeRearAxisZ.commandConfiguration.phasing.profileReference := 0;
   cmMendrelCathodeRearAxisZ.commandConfiguration.phasing.phasingDistance := 0.0;
   cmMendrelCathodeRearAxisZ.commandConfiguration.phasing.startPosition := 0.0;
   cmMendrelCathodeRearAxisZ.commandConfiguration.phasing.direction := 3;
   cmMendrelCathodeRearAxisZ.commandConfiguration.phasing.phaseAbsolute := TRUE;
   cmMendrelCathodeRearAxisZ.commandConfiguration.phasing.phaseShiftChangeOnTheFly := FALSE;
   cmMendrelCathodeRearAxisZ.commandConfiguration.offset.offset := 0.0;
   cmMendrelCathodeRearAxisZ.commandConfiguration.offset.profileReference := 1;
   cmMendrelCathodeRearAxisZ.commandConfiguration.offset.offsetDistance := 0.0;
   cmMendrelCathodeRearAxisZ.commandConfiguration.offset.startPosition := 0.0;
   cmMendrelCathodeRearAxisZ.commandConfiguration.offset.direction := 3;
   cmMendrelCathodeRearAxisZ.commandConfiguration.offset.offsetAbsolute := TRUE;
   cmMendrelCathodeRearAxisZ.commandConfiguration.offset.offsetChangeOnTheFly := FALSE;
   cmMendrelCathodeRearAxisZ.commands.enableAxis := FALSE;
   cmMendrelCathodeRearAxisZ.commands.resetAxis := FALSE;
   cmMendrelCathodeRearAxisZ.commands.openBrake := FALSE;
   cmMendrelCathodeRearAxisZ.commands.jogForward := FALSE;
   cmMendrelCathodeRearAxisZ.commands.jogBackward := FALSE;
   cmMendrelCathodeRearAxisZ.commands.moveVelocity := FALSE;
   cmMendrelCathodeRearAxisZ.commands.stop := FALSE;
   cmMendrelCathodeRearAxisZ.commands.fastStop := FALSE;
   cmMendrelCathodeRearAxisZ.commands.torqueLimiting := FALSE;
   cmMendrelCathodeRearAxisZ.commands.homing := FALSE;
   cmMendrelCathodeRearAxisZ.commands.posRelative := FALSE;
   cmMendrelCathodeRearAxisZ.commands.posAbsolute := FALSE;
   cmMendrelCathodeRearAxisZ.commands.posSuperimposed := FALSE;
   cmMendrelCathodeRearAxisZ.commands.haltSuperimposed := FALSE;
   cmMendrelCathodeRearAxisZ.commands.selectSetPosition := -1;
   cmMendrelCathodeRearAxisZ.commands.reset := FALSE;
   cmMendrelCathodeRearAxisZ.monitoring.valid := FALSE;
   cmMendrelCathodeRearAxisZ.monitoring.busy := TRUE;
   cmMendrelCathodeRearAxisZ.monitoring.error := TRUE;
   cmMendrelCathodeRearAxisZ.monitoring.status := 16#8600;
   cmMendrelCathodeRearAxisZ.monitoring.subfunctionStatus := 16#8001;
   cmMendrelCathodeRearAxisZ.monitoring.axisEnabled := FALSE;
   cmMendrelCathodeRearAxisZ.monitoring.resetActive := FALSE;
   cmMendrelCathodeRearAxisZ.monitoring.inVelocity := FALSE;
   cmMendrelCathodeRearAxisZ.monitoring.inLimitation := FALSE;
   cmMendrelCathodeRearAxisZ.monitoring.inClamping := FALSE;
   cmMendrelCathodeRearAxisZ.monitoring.startSync := FALSE;
   cmMendrelCathodeRearAxisZ.monitoring.inSync := FALSE;
   cmMendrelCathodeRearAxisZ.monitoring.inSimulation := FALSE;
   cmMendrelCathodeRearAxisZ.monitoring.jogSelected := FALSE;
   cmMendrelCathodeRearAxisZ.monitoring.moveVelocitySelected := FALSE;
   cmMendrelCathodeRearAxisZ.monitoring.stopSelected := FALSE;
   cmMendrelCathodeRearAxisZ.monitoring.fastStopSelected := FALSE;
   cmMendrelCathodeRearAxisZ.monitoring.torqueLimitingSelected := FALSE;
   cmMendrelCathodeRearAxisZ.monitoring.homingSelected := FALSE;
   cmMendrelCathodeRearAxisZ.monitoring.posRelativeSelected := FALSE;
   cmMendrelCathodeRearAxisZ.monitoring.posAbsoluteSelected := FALSE;
   cmMendrelCathodeRearAxisZ.monitoring.posSuperimposedSelected := FALSE;
   cmMendrelCathodeRearAxisZ.monitoring.haltSuperimposedSelected := FALSE;
   cmMendrelCathodeRearAxisZ.monitoring.commandBusy := FALSE;
   cmMendrelCathodeRearAxisZ.monitoring.commandDone := FALSE;
   cmMendrelCathodeRearAxisZ.monitoring.commandAborted := FALSE;
   cmMendrelCathodeRearAxisZ.monitoring.homingCommandBusy := FALSE;
   cmMendrelCathodeRearAxisZ.monitoring.homingCommandDone := FALSE;
   cmMendrelCathodeRearAxisZ.monitoring.homingCommandAborted := FALSE;
   cmMendrelCathodeRearAxisZ.monitoring.superimposedBusy := FALSE;
   cmMendrelCathodeRearAxisZ.monitoring.superimposedDone := FALSE;
   cmMendrelCathodeRearAxisZ.monitoring.superimposedAborted := FALSE;
   cmMendrelCathodeRearAxisZ.monitoring.actualPosition := 13.339;
   cmMendrelCathodeRearAxisZ.monitoring.actualSpeed := 0.0;
   cmMendrelCathodeRearAxisZ.monitoring.speedUnit := 1062;
   cmMendrelCathodeRearAxisZ.monitoring.positionUnit := 1013;
   cmMendrelCathodeRearAxisZ.monitoring.axisType := 1;
   cmMendrelCathodeRearAxisZ.monitoring.interlockGeneralOut := TRUE;
   cmMendrelCathodeRearAxisZ.monitoring.interlockJogForwardOut := TRUE;
   cmMendrelCathodeRearAxisZ.monitoring.interlockJogBackwardOut := TRUE;
   cmStackTableAxisZ.commandConfiguration.generalSettings.stopOnError := TRUE;
   cmStackTableAxisZ.commandConfiguration.generalSettings.resetWithRestart := FALSE;
   cmStackTableAxisZ.commandConfiguration.generalSettings.abortWaitingSyncCmd := TRUE;
   cmStackTableAxisZ.commandConfiguration.power.startMode := 1;
   cmStackTableAxisZ.commandConfiguration.power.stopMode := 0;
   cmStackTableAxisZ.commandConfiguration.power.syncMotionSimulation := FALSE;
   cmStackTableAxisZ.commandConfiguration.power.syncMotionSimulationExtendedMode := -1;
   cmStackTableAxisZ.commandConfiguration.jog.velocity := 0.0;
   cmStackTableAxisZ.commandConfiguration.jog.acceleration := -1.0;
   cmStackTableAxisZ.commandConfiguration.jog.deceleration := -1.0;
   cmStackTableAxisZ.commandConfiguration.jog.jerk := -1.0;
   cmStackTableAxisZ.commandConfiguration.jog.positionControlled := TRUE;
   cmStackTableAxisZ.commandConfiguration.jog.increment := 0.0;
   cmStackTableAxisZ.commandConfiguration.jog.mode := 0;
   cmStackTableAxisZ.commandConfiguration.moveVelocity.velocity := 0.0;
   cmStackTableAxisZ.commandConfiguration.moveVelocity.acceleration := -1.0;
   cmStackTableAxisZ.commandConfiguration.moveVelocity.deceleration := -1.0;
   cmStackTableAxisZ.commandConfiguration.moveVelocity.jerk := -1.0;
   cmStackTableAxisZ.commandConfiguration.moveVelocity.direction := 0;
   cmStackTableAxisZ.commandConfiguration.moveVelocity.positionControlled := TRUE;
   cmStackTableAxisZ.commandConfiguration.moveVelocity.velocityChangeOnTheFly := FALSE;
   cmStackTableAxisZ.commandConfiguration.stop.deceleration := -1.0;
   cmStackTableAxisZ.commandConfiguration.stop.jerk := -1.0;
   cmStackTableAxisZ.commandConfiguration.stop.abortAcceleration := FALSE;
   cmStackTableAxisZ.commandConfiguration.fastStop.deceleration := -1.0;
   cmStackTableAxisZ.commandConfiguration.fastStop.jerk := -1.0;
   cmStackTableAxisZ.commandConfiguration.fastStop.abortAcceleration := FALSE;
   cmStackTableAxisZ.commandConfiguration.fastStop.replaceStopPossible := FALSE;
   cmStackTableAxisZ.commandConfiguration.torqueLimiting.limit := -1.0;
   cmStackTableAxisZ.commandConfiguration.torqueLimiting.mode := 0;
   cmStackTableAxisZ.commandConfiguration.homing.position := 0.0;
   cmStackTableAxisZ.commandConfiguration.homing.mode := 0;
   cmStackTableAxisZ.commandConfiguration.homing.sensor := 0;
   cmStackTableAxisZ.commandConfiguration.homing.extendedMode := -1;
   cmStackTableAxisZ.commandConfiguration.homing.extendedModeTorqueLimit := 0.0;
   cmStackTableAxisZ.commandConfiguration.homing.extendedModeTargetPosition := 0.0;
   cmStackTableAxisZ.commandConfiguration.posRelative.distance := 0.0;
   cmStackTableAxisZ.commandConfiguration.posRelative.velocity := -1.0;
   cmStackTableAxisZ.commandConfiguration.posRelative.acceleration := -1.0;
   cmStackTableAxisZ.commandConfiguration.posRelative.deceleration := -1.0;
   cmStackTableAxisZ.commandConfiguration.posRelative.jerk := -1.0;
   cmStackTableAxisZ.commandConfiguration.posRelative.direction := 0;
   cmStackTableAxisZ.commandConfiguration.posAbsolute.position := 0.0;
   cmStackTableAxisZ.commandConfiguration.posAbsolute.velocity := -1.0;
   cmStackTableAxisZ.commandConfiguration.posAbsolute.acceleration := -1.0;
   cmStackTableAxisZ.commandConfiguration.posAbsolute.deceleration := -1.0;
   cmStackTableAxisZ.commandConfiguration.posAbsolute.jerk := -1.0;
   cmStackTableAxisZ.commandConfiguration.posAbsolute.direction := 1;
   cmStackTableAxisZ.commandConfiguration.posAbsolute.positionChangeOnTheFly := FALSE;
   cmStackTableAxisZ.commandConfiguration.posAbsolute.velocityChangeOnTheFly := FALSE;
   cmStackTableAxisZ.commandConfiguration.posSuperimposed.distance := 0.0;
   cmStackTableAxisZ.commandConfiguration.posSuperimposed.velocityDiff := -1.0;
   cmStackTableAxisZ.commandConfiguration.posSuperimposed.acceleration := -1.0;
   cmStackTableAxisZ.commandConfiguration.posSuperimposed.deceleration := -1.0;
   cmStackTableAxisZ.commandConfiguration.posSuperimposed.jerk := -1.0;
   cmStackTableAxisZ.commandConfiguration.posSuperimposed.direction := 0;
   cmStackTableAxisZ.commandConfiguration.haltSuperimposed.deceleration := -1.0;
   cmStackTableAxisZ.commandConfiguration.haltSuperimposed.jerk := -1.0;
   cmStackTableAxisZ.commandConfiguration.haltSuperimposed.abortAcceleration := FALSE;
   cmStackTableAxisZ.commandConfiguration.gearInRelative.ratioNumerator := 1;
   cmStackTableAxisZ.commandConfiguration.gearInRelative.ratioDenominator := 1;
   cmStackTableAxisZ.commandConfiguration.gearInRelative.acceleration := -1.0;
   cmStackTableAxisZ.commandConfiguration.gearInRelative.deceleration := -1.0;
   cmStackTableAxisZ.commandConfiguration.gearInRelative.jerk := -1.0;
   cmStackTableAxisZ.commandConfiguration.gearInRelative.ratioChangeOnTheFly := FALSE;
   cmStackTableAxisZ.commandConfiguration.gearInAbsolute.ratioNumerator := 1;
   cmStackTableAxisZ.commandConfiguration.gearInAbsolute.ratioDenominator := 1;
   cmStackTableAxisZ.commandConfiguration.gearInAbsolute.masterSyncPosition := 0.0;
   cmStackTableAxisZ.commandConfiguration.gearInAbsolute.slaveSyncPosition := 0.0;
   cmStackTableAxisZ.commandConfiguration.gearInAbsolute.syncProfileReference := 1;
   cmStackTableAxisZ.commandConfiguration.gearInAbsolute.masterStartDistance := 0.0;
   cmStackTableAxisZ.commandConfiguration.gearInAbsolute.velocity := -1.0;
   cmStackTableAxisZ.commandConfiguration.gearInAbsolute.acceleration := -1.0;
   cmStackTableAxisZ.commandConfiguration.gearInAbsolute.deceleration := -1.0;
   cmStackTableAxisZ.commandConfiguration.gearInAbsolute.jerk := -1.0;
   cmStackTableAxisZ.commandConfiguration.gearInAbsolute.syncDirection := 1;
   cmStackTableAxisZ.commandConfiguration.gearInAbsolute.ratioChangeOnTheFly := FALSE;
   cmStackTableAxisZ.commandConfiguration.gearInVelocity.continuousUpdate := FALSE;
   cmStackTableAxisZ.commandConfiguration.gearInVelocity.ratioNumerator := 1;
   cmStackTableAxisZ.commandConfiguration.gearInVelocity.ratioDenominator := 1;
   cmStackTableAxisZ.commandConfiguration.gearInVelocity.acceleration := -1.0;
   cmStackTableAxisZ.commandConfiguration.gearInVelocity.deceleration := -1.0;
   cmStackTableAxisZ.commandConfiguration.gearInVelocity.jerk := -1.0;
   cmStackTableAxisZ.commandConfiguration.gearInVelocity.positionControlled := FALSE;
   cmStackTableAxisZ.commandConfiguration.camIn.masterOffset := 0.0;
   cmStackTableAxisZ.commandConfiguration.camIn.slaveOffset := 0.0;
   cmStackTableAxisZ.commandConfiguration.camIn.masterScaling := 1.0;
   cmStackTableAxisZ.commandConfiguration.camIn.slaveScaling := 1.0;
   cmStackTableAxisZ.commandConfiguration.camIn.masterSyncPosition := 0.0;
   cmStackTableAxisZ.commandConfiguration.camIn.syncProfileReference := 1;
   cmStackTableAxisZ.commandConfiguration.camIn.masterStartDistance := 0.0;
   cmStackTableAxisZ.commandConfiguration.camIn.velocity := -1.0;
   cmStackTableAxisZ.commandConfiguration.camIn.acceleration := -1.0;
   cmStackTableAxisZ.commandConfiguration.camIn.deceleration := -1.0;
   cmStackTableAxisZ.commandConfiguration.camIn.jerk := -1.0;
   cmStackTableAxisZ.commandConfiguration.camIn.applicationMode := 0;
   cmStackTableAxisZ.commandConfiguration.camIn.syncDirection := 1;
   cmStackTableAxisZ.commandConfiguration.gearOutCamOut.slavePosition := 0.0;
   cmStackTableAxisZ.commandConfiguration.gearOutCamOut.syncProfileReference := 1;
   cmStackTableAxisZ.commandConfiguration.gearOutCamOut.masterStopDistance := 0.0;
   cmStackTableAxisZ.commandConfiguration.gearOutCamOut.deceleration := -1.0;
   cmStackTableAxisZ.commandConfiguration.gearOutCamOut.jerk := -1.0;
   cmStackTableAxisZ.commandConfiguration.gearOutCamOut.syncOutDirection := 3;
   cmStackTableAxisZ.commandConfiguration.gearOutCamOut.gearOutCamOutMode := -1;
   cmStackTableAxisZ.commandConfiguration.phasing.phaseShift := 0.0;
   cmStackTableAxisZ.commandConfiguration.phasing.velocity := -1.0;
   cmStackTableAxisZ.commandConfiguration.phasing.acceleration := -1.0;
   cmStackTableAxisZ.commandConfiguration.phasing.deceleration := -1.0;
   cmStackTableAxisZ.commandConfiguration.phasing.jerk := -1.0;
   cmStackTableAxisZ.commandConfiguration.phasing.profileReference := 0;
   cmStackTableAxisZ.commandConfiguration.phasing.phasingDistance := 0.0;
   cmStackTableAxisZ.commandConfiguration.phasing.startPosition := 0.0;
   cmStackTableAxisZ.commandConfiguration.phasing.direction := 3;
   cmStackTableAxisZ.commandConfiguration.phasing.phaseAbsolute := TRUE;
   cmStackTableAxisZ.commandConfiguration.phasing.phaseShiftChangeOnTheFly := FALSE;
   cmStackTableAxisZ.commandConfiguration.offset.offset := 0.0;
   cmStackTableAxisZ.commandConfiguration.offset.profileReference := 1;
   cmStackTableAxisZ.commandConfiguration.offset.offsetDistance := 0.0;
   cmStackTableAxisZ.commandConfiguration.offset.startPosition := 0.0;
   cmStackTableAxisZ.commandConfiguration.offset.direction := 3;
   cmStackTableAxisZ.commandConfiguration.offset.offsetAbsolute := TRUE;
   cmStackTableAxisZ.commandConfiguration.offset.offsetChangeOnTheFly := FALSE;
   cmStackTableAxisZ.commands.enableAxis := FALSE;
   cmStackTableAxisZ.commands.resetAxis := FALSE;
   cmStackTableAxisZ.commands.openBrake := FALSE;
   cmStackTableAxisZ.commands.jogForward := FALSE;
   cmStackTableAxisZ.commands.jogBackward := FALSE;
   cmStackTableAxisZ.commands.moveVelocity := FALSE;
   cmStackTableAxisZ.commands.stop := FALSE;
   cmStackTableAxisZ.commands.fastStop := FALSE;
   cmStackTableAxisZ.commands.torqueLimiting := FALSE;
   cmStackTableAxisZ.commands.homing := FALSE;
   cmStackTableAxisZ.commands.posRelative := FALSE;
   cmStackTableAxisZ.commands.posAbsolute := FALSE;
   cmStackTableAxisZ.commands.posSuperimposed := FALSE;
   cmStackTableAxisZ.commands.haltSuperimposed := FALSE;
   cmStackTableAxisZ.commands.selectSetPosition := -1;
   cmStackTableAxisZ.commands.reset := FALSE;
   cmStackTableAxisZ.monitoring.valid := FALSE;
   cmStackTableAxisZ.monitoring.busy := TRUE;
   cmStackTableAxisZ.monitoring.error := TRUE;
   cmStackTableAxisZ.monitoring.status := 16#8600;
   cmStackTableAxisZ.monitoring.subfunctionStatus := 16#8001;
   cmStackTableAxisZ.monitoring.axisEnabled := FALSE;
   cmStackTableAxisZ.monitoring.resetActive := FALSE;
   cmStackTableAxisZ.monitoring.inVelocity := FALSE;
   cmStackTableAxisZ.monitoring.inLimitation := FALSE;
   cmStackTableAxisZ.monitoring.inClamping := FALSE;
   cmStackTableAxisZ.monitoring.startSync := FALSE;
   cmStackTableAxisZ.monitoring.inSync := FALSE;
   cmStackTableAxisZ.monitoring.inSimulation := FALSE;
   cmStackTableAxisZ.monitoring.jogSelected := FALSE;
   cmStackTableAxisZ.monitoring.moveVelocitySelected := FALSE;
   cmStackTableAxisZ.monitoring.stopSelected := FALSE;
   cmStackTableAxisZ.monitoring.fastStopSelected := FALSE;
   cmStackTableAxisZ.monitoring.torqueLimitingSelected := FALSE;
   cmStackTableAxisZ.monitoring.homingSelected := FALSE;
   cmStackTableAxisZ.monitoring.posRelativeSelected := FALSE;
   cmStackTableAxisZ.monitoring.posAbsoluteSelected := FALSE;
   cmStackTableAxisZ.monitoring.posSuperimposedSelected := FALSE;
   cmStackTableAxisZ.monitoring.haltSuperimposedSelected := FALSE;
   cmStackTableAxisZ.monitoring.commandBusy := FALSE;
   cmStackTableAxisZ.monitoring.commandDone := FALSE;
   cmStackTableAxisZ.monitoring.commandAborted := FALSE;
   cmStackTableAxisZ.monitoring.homingCommandBusy := FALSE;
   cmStackTableAxisZ.monitoring.homingCommandDone := FALSE;
   cmStackTableAxisZ.monitoring.homingCommandAborted := FALSE;
   cmStackTableAxisZ.monitoring.superimposedBusy := FALSE;
   cmStackTableAxisZ.monitoring.superimposedDone := FALSE;
   cmStackTableAxisZ.monitoring.superimposedAborted := FALSE;
   cmStackTableAxisZ.monitoring.actualPosition := -20.199;
   cmStackTableAxisZ.monitoring.actualSpeed := 0.0;
   cmStackTableAxisZ.monitoring.speedUnit := 1062;
   cmStackTableAxisZ.monitoring.positionUnit := 1013;
   cmStackTableAxisZ.monitoring.axisType := 1;
   cmStackTableAxisZ.monitoring.interlockGeneralOut := FALSE;
   cmStackTableAxisZ.monitoring.interlockJogForwardOut := TRUE;
   cmStackTableAxisZ.monitoring.interlockJogBackwardOut := TRUE;
   cmStackTableOutFrontAxisZ.commandConfiguration.generalSettings.stopOnError := TRUE;
   cmStackTableOutFrontAxisZ.commandConfiguration.generalSettings.resetWithRestart := FALSE;
   cmStackTableOutFrontAxisZ.commandConfiguration.generalSettings.abortWaitingSyncCmd := TRUE;
   cmStackTableOutFrontAxisZ.commandConfiguration.power.startMode := 1;
   cmStackTableOutFrontAxisZ.commandConfiguration.power.stopMode := 0;
   cmStackTableOutFrontAxisZ.commandConfiguration.power.syncMotionSimulation := FALSE;
   cmStackTableOutFrontAxisZ.commandConfiguration.power.syncMotionSimulationExtendedMode := -1;
   cmStackTableOutFrontAxisZ.commandConfiguration.jog.velocity := 0.0;
   cmStackTableOutFrontAxisZ.commandConfiguration.jog.acceleration := -1.0;
   cmStackTableOutFrontAxisZ.commandConfiguration.jog.deceleration := -1.0;
   cmStackTableOutFrontAxisZ.commandConfiguration.jog.jerk := -1.0;
   cmStackTableOutFrontAxisZ.commandConfiguration.jog.positionControlled := TRUE;
   cmStackTableOutFrontAxisZ.commandConfiguration.jog.increment := 0.0;
   cmStackTableOutFrontAxisZ.commandConfiguration.jog.mode := 0;
   cmStackTableOutFrontAxisZ.commandConfiguration.moveVelocity.velocity := 0.0;
   cmStackTableOutFrontAxisZ.commandConfiguration.moveVelocity.acceleration := -1.0;
   cmStackTableOutFrontAxisZ.commandConfiguration.moveVelocity.deceleration := -1.0;
   cmStackTableOutFrontAxisZ.commandConfiguration.moveVelocity.jerk := -1.0;
   cmStackTableOutFrontAxisZ.commandConfiguration.moveVelocity.direction := 0;
   cmStackTableOutFrontAxisZ.commandConfiguration.moveVelocity.positionControlled := TRUE;
   cmStackTableOutFrontAxisZ.commandConfiguration.moveVelocity.velocityChangeOnTheFly := FALSE;
   cmStackTableOutFrontAxisZ.commandConfiguration.stop.deceleration := -1.0;
   cmStackTableOutFrontAxisZ.commandConfiguration.stop.jerk := -1.0;
   cmStackTableOutFrontAxisZ.commandConfiguration.stop.abortAcceleration := FALSE;
   cmStackTableOutFrontAxisZ.commandConfiguration.fastStop.deceleration := -1.0;
   cmStackTableOutFrontAxisZ.commandConfiguration.fastStop.jerk := -1.0;
   cmStackTableOutFrontAxisZ.commandConfiguration.fastStop.abortAcceleration := FALSE;
   cmStackTableOutFrontAxisZ.commandConfiguration.fastStop.replaceStopPossible := FALSE;
   cmStackTableOutFrontAxisZ.commandConfiguration.torqueLimiting.limit := -1.0;
   cmStackTableOutFrontAxisZ.commandConfiguration.torqueLimiting.mode := 0;
   cmStackTableOutFrontAxisZ.commandConfiguration.homing.position := 0.0;
   cmStackTableOutFrontAxisZ.commandConfiguration.homing.mode := 0;
   cmStackTableOutFrontAxisZ.commandConfiguration.homing.sensor := 0;
   cmStackTableOutFrontAxisZ.commandConfiguration.homing.extendedMode := -1;
   cmStackTableOutFrontAxisZ.commandConfiguration.homing.extendedModeTorqueLimit := 0.0;
   cmStackTableOutFrontAxisZ.commandConfiguration.homing.extendedModeTargetPosition := 0.0;
   cmStackTableOutFrontAxisZ.commandConfiguration.posRelative.distance := 0.0;
   cmStackTableOutFrontAxisZ.commandConfiguration.posRelative.velocity := -1.0;
   cmStackTableOutFrontAxisZ.commandConfiguration.posRelative.acceleration := -1.0;
   cmStackTableOutFrontAxisZ.commandConfiguration.posRelative.deceleration := -1.0;
   cmStackTableOutFrontAxisZ.commandConfiguration.posRelative.jerk := -1.0;
   cmStackTableOutFrontAxisZ.commandConfiguration.posRelative.direction := 0;
   cmStackTableOutFrontAxisZ.commandConfiguration.posAbsolute.position := 0.0;
   cmStackTableOutFrontAxisZ.commandConfiguration.posAbsolute.velocity := -1.0;
   cmStackTableOutFrontAxisZ.commandConfiguration.posAbsolute.acceleration := -1.0;
   cmStackTableOutFrontAxisZ.commandConfiguration.posAbsolute.deceleration := -1.0;
   cmStackTableOutFrontAxisZ.commandConfiguration.posAbsolute.jerk := -1.0;
   cmStackTableOutFrontAxisZ.commandConfiguration.posAbsolute.direction := 1;
   cmStackTableOutFrontAxisZ.commandConfiguration.posAbsolute.positionChangeOnTheFly := FALSE;
   cmStackTableOutFrontAxisZ.commandConfiguration.posAbsolute.velocityChangeOnTheFly := FALSE;
   cmStackTableOutFrontAxisZ.commandConfiguration.posSuperimposed.distance := 0.0;
   cmStackTableOutFrontAxisZ.commandConfiguration.posSuperimposed.velocityDiff := -1.0;
   cmStackTableOutFrontAxisZ.commandConfiguration.posSuperimposed.acceleration := -1.0;
   cmStackTableOutFrontAxisZ.commandConfiguration.posSuperimposed.deceleration := -1.0;
   cmStackTableOutFrontAxisZ.commandConfiguration.posSuperimposed.jerk := -1.0;
   cmStackTableOutFrontAxisZ.commandConfiguration.posSuperimposed.direction := 0;
   cmStackTableOutFrontAxisZ.commandConfiguration.haltSuperimposed.deceleration := -1.0;
   cmStackTableOutFrontAxisZ.commandConfiguration.haltSuperimposed.jerk := -1.0;
   cmStackTableOutFrontAxisZ.commandConfiguration.haltSuperimposed.abortAcceleration := FALSE;
   cmStackTableOutFrontAxisZ.commandConfiguration.gearInRelative.ratioNumerator := 1;
   cmStackTableOutFrontAxisZ.commandConfiguration.gearInRelative.ratioDenominator := 1;
   cmStackTableOutFrontAxisZ.commandConfiguration.gearInRelative.acceleration := -1.0;
   cmStackTableOutFrontAxisZ.commandConfiguration.gearInRelative.deceleration := -1.0;
   cmStackTableOutFrontAxisZ.commandConfiguration.gearInRelative.jerk := -1.0;
   cmStackTableOutFrontAxisZ.commandConfiguration.gearInRelative.ratioChangeOnTheFly := FALSE;
   cmStackTableOutFrontAxisZ.commandConfiguration.gearInAbsolute.ratioNumerator := 1;
   cmStackTableOutFrontAxisZ.commandConfiguration.gearInAbsolute.ratioDenominator := 1;
   cmStackTableOutFrontAxisZ.commandConfiguration.gearInAbsolute.masterSyncPosition := 0.0;
   cmStackTableOutFrontAxisZ.commandConfiguration.gearInAbsolute.slaveSyncPosition := 0.0;
   cmStackTableOutFrontAxisZ.commandConfiguration.gearInAbsolute.syncProfileReference := 1;
   cmStackTableOutFrontAxisZ.commandConfiguration.gearInAbsolute.masterStartDistance := 0.0;
   cmStackTableOutFrontAxisZ.commandConfiguration.gearInAbsolute.velocity := -1.0;
   cmStackTableOutFrontAxisZ.commandConfiguration.gearInAbsolute.acceleration := -1.0;
   cmStackTableOutFrontAxisZ.commandConfiguration.gearInAbsolute.deceleration := -1.0;
   cmStackTableOutFrontAxisZ.commandConfiguration.gearInAbsolute.jerk := -1.0;
   cmStackTableOutFrontAxisZ.commandConfiguration.gearInAbsolute.syncDirection := 1;
   cmStackTableOutFrontAxisZ.commandConfiguration.gearInAbsolute.ratioChangeOnTheFly := FALSE;
   cmStackTableOutFrontAxisZ.commandConfiguration.gearInVelocity.continuousUpdate := FALSE;
   cmStackTableOutFrontAxisZ.commandConfiguration.gearInVelocity.ratioNumerator := 1;
   cmStackTableOutFrontAxisZ.commandConfiguration.gearInVelocity.ratioDenominator := 1;
   cmStackTableOutFrontAxisZ.commandConfiguration.gearInVelocity.acceleration := -1.0;
   cmStackTableOutFrontAxisZ.commandConfiguration.gearInVelocity.deceleration := -1.0;
   cmStackTableOutFrontAxisZ.commandConfiguration.gearInVelocity.jerk := -1.0;
   cmStackTableOutFrontAxisZ.commandConfiguration.gearInVelocity.positionControlled := FALSE;
   cmStackTableOutFrontAxisZ.commandConfiguration.camIn.masterOffset := 0.0;
   cmStackTableOutFrontAxisZ.commandConfiguration.camIn.slaveOffset := 0.0;
   cmStackTableOutFrontAxisZ.commandConfiguration.camIn.masterScaling := 1.0;
   cmStackTableOutFrontAxisZ.commandConfiguration.camIn.slaveScaling := 1.0;
   cmStackTableOutFrontAxisZ.commandConfiguration.camIn.masterSyncPosition := 0.0;
   cmStackTableOutFrontAxisZ.commandConfiguration.camIn.syncProfileReference := 1;
   cmStackTableOutFrontAxisZ.commandConfiguration.camIn.masterStartDistance := 0.0;
   cmStackTableOutFrontAxisZ.commandConfiguration.camIn.velocity := -1.0;
   cmStackTableOutFrontAxisZ.commandConfiguration.camIn.acceleration := -1.0;
   cmStackTableOutFrontAxisZ.commandConfiguration.camIn.deceleration := -1.0;
   cmStackTableOutFrontAxisZ.commandConfiguration.camIn.jerk := -1.0;
   cmStackTableOutFrontAxisZ.commandConfiguration.camIn.applicationMode := 0;
   cmStackTableOutFrontAxisZ.commandConfiguration.camIn.syncDirection := 1;
   cmStackTableOutFrontAxisZ.commandConfiguration.gearOutCamOut.slavePosition := 0.0;
   cmStackTableOutFrontAxisZ.commandConfiguration.gearOutCamOut.syncProfileReference := 1;
   cmStackTableOutFrontAxisZ.commandConfiguration.gearOutCamOut.masterStopDistance := 0.0;
   cmStackTableOutFrontAxisZ.commandConfiguration.gearOutCamOut.deceleration := -1.0;
   cmStackTableOutFrontAxisZ.commandConfiguration.gearOutCamOut.jerk := -1.0;
   cmStackTableOutFrontAxisZ.commandConfiguration.gearOutCamOut.syncOutDirection := 3;
   cmStackTableOutFrontAxisZ.commandConfiguration.gearOutCamOut.gearOutCamOutMode := -1;
   cmStackTableOutFrontAxisZ.commandConfiguration.phasing.phaseShift := 0.0;
   cmStackTableOutFrontAxisZ.commandConfiguration.phasing.velocity := -1.0;
   cmStackTableOutFrontAxisZ.commandConfiguration.phasing.acceleration := -1.0;
   cmStackTableOutFrontAxisZ.commandConfiguration.phasing.deceleration := -1.0;
   cmStackTableOutFrontAxisZ.commandConfiguration.phasing.jerk := -1.0;
   cmStackTableOutFrontAxisZ.commandConfiguration.phasing.profileReference := 0;
   cmStackTableOutFrontAxisZ.commandConfiguration.phasing.phasingDistance := 0.0;
   cmStackTableOutFrontAxisZ.commandConfiguration.phasing.startPosition := 0.0;
   cmStackTableOutFrontAxisZ.commandConfiguration.phasing.direction := 3;
   cmStackTableOutFrontAxisZ.commandConfiguration.phasing.phaseAbsolute := TRUE;
   cmStackTableOutFrontAxisZ.commandConfiguration.phasing.phaseShiftChangeOnTheFly := FALSE;
   cmStackTableOutFrontAxisZ.commandConfiguration.offset.offset := 0.0;
   cmStackTableOutFrontAxisZ.commandConfiguration.offset.profileReference := 1;
   cmStackTableOutFrontAxisZ.commandConfiguration.offset.offsetDistance := 0.0;
   cmStackTableOutFrontAxisZ.commandConfiguration.offset.startPosition := 0.0;
   cmStackTableOutFrontAxisZ.commandConfiguration.offset.direction := 3;
   cmStackTableOutFrontAxisZ.commandConfiguration.offset.offsetAbsolute := TRUE;
   cmStackTableOutFrontAxisZ.commandConfiguration.offset.offsetChangeOnTheFly := FALSE;
   cmStackTableOutFrontAxisZ.commands.enableAxis := FALSE;
   cmStackTableOutFrontAxisZ.commands.resetAxis := FALSE;
   cmStackTableOutFrontAxisZ.commands.openBrake := FALSE;
   cmStackTableOutFrontAxisZ.commands.jogForward := FALSE;
   cmStackTableOutFrontAxisZ.commands.jogBackward := FALSE;
   cmStackTableOutFrontAxisZ.commands.moveVelocity := FALSE;
   cmStackTableOutFrontAxisZ.commands.stop := FALSE;
   cmStackTableOutFrontAxisZ.commands.fastStop := FALSE;
   cmStackTableOutFrontAxisZ.commands.torqueLimiting := FALSE;
   cmStackTableOutFrontAxisZ.commands.homing := FALSE;
   cmStackTableOutFrontAxisZ.commands.posRelative := FALSE;
   cmStackTableOutFrontAxisZ.commands.posAbsolute := FALSE;
   cmStackTableOutFrontAxisZ.commands.posSuperimposed := FALSE;
   cmStackTableOutFrontAxisZ.commands.haltSuperimposed := FALSE;
   cmStackTableOutFrontAxisZ.commands.selectSetPosition := -1;
   cmStackTableOutFrontAxisZ.commands.reset := FALSE;
   cmStackTableOutFrontAxisZ.monitoring.valid := FALSE;
   cmStackTableOutFrontAxisZ.monitoring.busy := TRUE;
   cmStackTableOutFrontAxisZ.monitoring.error := TRUE;
   cmStackTableOutFrontAxisZ.monitoring.status := 16#8600;
   cmStackTableOutFrontAxisZ.monitoring.subfunctionStatus := 16#8001;
   cmStackTableOutFrontAxisZ.monitoring.axisEnabled := FALSE;
   cmStackTableOutFrontAxisZ.monitoring.resetActive := FALSE;
   cmStackTableOutFrontAxisZ.monitoring.inVelocity := FALSE;
   cmStackTableOutFrontAxisZ.monitoring.inLimitation := FALSE;
   cmStackTableOutFrontAxisZ.monitoring.inClamping := FALSE;
   cmStackTableOutFrontAxisZ.monitoring.startSync := FALSE;
   cmStackTableOutFrontAxisZ.monitoring.inSync := FALSE;
   cmStackTableOutFrontAxisZ.monitoring.inSimulation := FALSE;
   cmStackTableOutFrontAxisZ.monitoring.jogSelected := FALSE;
   cmStackTableOutFrontAxisZ.monitoring.moveVelocitySelected := FALSE;
   cmStackTableOutFrontAxisZ.monitoring.stopSelected := FALSE;
   cmStackTableOutFrontAxisZ.monitoring.fastStopSelected := FALSE;
   cmStackTableOutFrontAxisZ.monitoring.torqueLimitingSelected := FALSE;
   cmStackTableOutFrontAxisZ.monitoring.homingSelected := FALSE;
   cmStackTableOutFrontAxisZ.monitoring.posRelativeSelected := FALSE;
   cmStackTableOutFrontAxisZ.monitoring.posAbsoluteSelected := FALSE;
   cmStackTableOutFrontAxisZ.monitoring.posSuperimposedSelected := FALSE;
   cmStackTableOutFrontAxisZ.monitoring.haltSuperimposedSelected := FALSE;
   cmStackTableOutFrontAxisZ.monitoring.commandBusy := FALSE;
   cmStackTableOutFrontAxisZ.monitoring.commandDone := FALSE;
   cmStackTableOutFrontAxisZ.monitoring.commandAborted := FALSE;
   cmStackTableOutFrontAxisZ.monitoring.homingCommandBusy := FALSE;
   cmStackTableOutFrontAxisZ.monitoring.homingCommandDone := FALSE;
   cmStackTableOutFrontAxisZ.monitoring.homingCommandAborted := FALSE;
   cmStackTableOutFrontAxisZ.monitoring.superimposedBusy := FALSE;
   cmStackTableOutFrontAxisZ.monitoring.superimposedDone := FALSE;
   cmStackTableOutFrontAxisZ.monitoring.superimposedAborted := FALSE;
   cmStackTableOutFrontAxisZ.monitoring.actualPosition := -14.802;
   cmStackTableOutFrontAxisZ.monitoring.actualSpeed := 0.0;
   cmStackTableOutFrontAxisZ.monitoring.speedUnit := 1062;
   cmStackTableOutFrontAxisZ.monitoring.positionUnit := 1013;
   cmStackTableOutFrontAxisZ.monitoring.axisType := 1;
   cmStackTableOutFrontAxisZ.monitoring.interlockGeneralOut := TRUE;
   cmStackTableOutFrontAxisZ.monitoring.interlockJogForwardOut := TRUE;
   cmStackTableOutFrontAxisZ.monitoring.interlockJogBackwardOut := TRUE;
   cmMendrelAnodeRearClamp.commands.commandHomePos := FALSE;
   cmMendrelAnodeRearClamp.commands.commandWorkPos := FALSE;
   cmMendrelAnodeRearClamp.commands.reset := FALSE;
   cmMendrelAnodeRearClamp.monitoring.valid := TRUE;
   cmMendrelAnodeRearClamp.monitoring.busy := TRUE;
   cmMendrelAnodeRearClamp.monitoring.error := FALSE;
   cmMendrelAnodeRearClamp.monitoring.status := 16#7003;
   cmMendrelAnodeRearClamp.monitoring.inHomePos := FALSE;
   cmMendrelAnodeRearClamp.monitoring.inWorkPos := FALSE;
   cmMendrelAnodeRearClamp.monitoring.interlockWorkPosOut := TRUE;
   cmMendrelAnodeRearClamp.monitoring.interlockHomePosOut := TRUE;
   cmMendrelCathodeFrontClamp.commands.commandHomePos := FALSE;
   cmMendrelCathodeFrontClamp.commands.commandWorkPos := FALSE;
   cmMendrelCathodeFrontClamp.commands.reset := FALSE;
   cmMendrelCathodeFrontClamp.monitoring.valid := TRUE;
   cmMendrelCathodeFrontClamp.monitoring.busy := TRUE;
   cmMendrelCathodeFrontClamp.monitoring.error := FALSE;
   cmMendrelCathodeFrontClamp.monitoring.status := 16#7003;
   cmMendrelCathodeFrontClamp.monitoring.inHomePos := FALSE;
   cmMendrelCathodeFrontClamp.monitoring.inWorkPos := FALSE;
   cmMendrelCathodeFrontClamp.monitoring.interlockWorkPosOut := TRUE;
   cmMendrelCathodeFrontClamp.monitoring.interlockHomePosOut := TRUE;
   cmMendrelCathodeRearClamp.commands.commandHomePos := FALSE;
   cmMendrelCathodeRearClamp.commands.commandWorkPos := FALSE;
   cmMendrelCathodeRearClamp.commands.reset := FALSE;
   cmMendrelCathodeRearClamp.monitoring.valid := TRUE;
   cmMendrelCathodeRearClamp.monitoring.busy := TRUE;
   cmMendrelCathodeRearClamp.monitoring.error := FALSE;
   cmMendrelCathodeRearClamp.monitoring.status := 16#7003;
   cmMendrelCathodeRearClamp.monitoring.inHomePos := FALSE;
   cmMendrelCathodeRearClamp.monitoring.inWorkPos := FALSE;
   cmMendrelCathodeRearClamp.monitoring.interlockWorkPosOut := TRUE;
   cmMendrelCathodeRearClamp.monitoring.interlockHomePosOut := TRUE;
   cmStackTableVaccum.commands.commandHomePos := FALSE;
   cmStackTableVaccum.commands.commandWorkPos := FALSE;
   cmStackTableVaccum.commands.reset := FALSE;
   cmStackTableVaccum.monitoring.valid := TRUE;
   cmStackTableVaccum.monitoring.busy := TRUE;
   cmStackTableVaccum.monitoring.error := FALSE;
   cmStackTableVaccum.monitoring.status := 16#7003;
   cmStackTableVaccum.monitoring.inHomePos := FALSE;
   cmStackTableVaccum.monitoring.inWorkPos := FALSE;
   cmStackTableVaccum.monitoring.interlockWorkPosOut := TRUE;
   cmStackTableVaccum.monitoring.interlockHomePosOut := TRUE;
   cmStackTableGapPadUpDown.commands.commandHomePos := FALSE;
   cmStackTableGapPadUpDown.commands.commandWorkPos := FALSE;
   cmStackTableGapPadUpDown.commands.reset := FALSE;
   cmStackTableGapPadUpDown.monitoring.valid := TRUE;
   cmStackTableGapPadUpDown.monitoring.busy := TRUE;
   cmStackTableGapPadUpDown.monitoring.error := FALSE;
   cmStackTableGapPadUpDown.monitoring.status := 16#7003;
   cmStackTableGapPadUpDown.monitoring.inHomePos := FALSE;
   cmStackTableGapPadUpDown.monitoring.inWorkPos := FALSE;
   cmStackTableGapPadUpDown.monitoring.interlockWorkPosOut := TRUE;
   cmStackTableGapPadUpDown.monitoring.interlockHomePosOut := TRUE;
END_DATA_BLOCK
